SUBAPPLICATION F (* Subapplication Type *)
  (* Standard: 61499-2 *)
  (* Version 1.0, 2025-02-12, franz *)
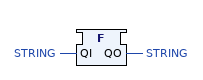
  VAR_INPUT
    QI : STRING; (* Input event qualifier *)
  END_VAR
  VAR_OUTPUT
    QO : STRING; (* Output event qualifier *)
  END_VAR
  DATA_CONNECTIONS
    QI TO QO;
  END_CONNECTIONS
END_SUBAPPLICATION
